{attribute 'pack_mode' := '2'}
TYPE ST_INSTANCE_STATE :
STRUCT
  State             : E_INSTANCE_STATE;
  Progress          : E_PROGRESS;

  QueueProcessCount : UINT; // sum of all queues in process
  StationCount      : UINT;
END_STRUCT
END_TYPE

(* stored: Version 1.1.0.1, ProductVersion 3.1.4026.18
   DUT ST_INSTANCE_STATE: Id {d222ca99-8d6b-4f76-9381-8da6e6918f58} *)
